# B&R Automation Studio project GettingStarted
Automation Studio 4.9

## Configuration NewConfiguration

CPU PC_any, AutomationRuntime G4.93, Build 4.1.2, Vc V4.72.6

### Task classes (Cpu.sw)
```
Cyclic#4:
  LampTest <- LampTest.prg
```

### Hardware
```
PC : PC_any v1.1.1.0 (OrderNumber=PC)
```

## Logical view

### Program Logical/LampTest (IEC)

#### Variables.var
```iecst
VAR
	Lamp : BOOL;
	Switch : BOOL;
END_VAR
```

#### Cyclic.ld
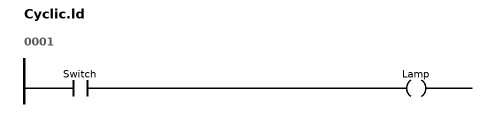
Ladder, written as Structured Text:
```iecst
PROGRAM _CYCLIC
(* Network 1 *)
Lamp := Switch;
END_PROGRAM
```

Listed in the project but not available here: Logical/Global.typ, Logical/Global.var, Logical/Libraries
